ABB RobotStudio station: Project1.rsstnx

Station Project1 (saved by RobotStudio 25.4.11475.0)
Controller IRB1200_5_90
  mechanical unit ROB_1: IRB1200_5_90_STD_03, 6 joints, base frame (0, 0, 0) mm
Layout (positions relative to the parent item):
  - IRB1200_5_90_STD_03 [mechanism, from %ABB.RobotStudio.Models.IRB1200%\IRB1200_5_90_STD_03.rslib] at (0, 0, 0) mm; joint values [0.0447, 0.6385, 0.2859, 0.007, 0.6807, -0.0091] (rad or m)
